FUNCTION_BLOCK FB_HE_SolidAttenuatorSlot EXTENDS FB_Fallible IMPLEMENTS I_HE_SolidAttenuatorSlot
VAR
    iFilter : I_HE_SolidAttenuatorFilter;
    eState : E_HE_SolidAttenuatorSlotState;
    bEnabled : BOOL;
END_VAR


METHOD FB_Init: BOOL
VAR_INPUT
    bInitRetains: BOOL; // TRUE: the retain variables are initialized (reset warm / reset cold)
    bInCopyCode: BOOL;  // TRUE: the instance will be copied to the copy code afterward (online change)

    Filter : I_HE_SolidAttenuatorFilter;
    State : E_HE_SolidAttenuatorSlotState;
    Enabled : BOOL;
END_VAR

iFilter := Filter;
eState := State;
bEnabled := Enabled;
END_METHOD


METHOD GetCenterPosition
VAR_INPUT
    CenterPosition : I_QuantityLREALPublic;
END_VAR

iFilter.GetCenterPosition(CenterPosition := CenterPosition);
END_METHOD


METHOD GetLength
VAR_INPUT
    Length : I_QuantityLREALPublic;
END_VAR

CASE eState OF
    E_HE_SolidAttenuatorSlotState.EMPTY:
        Length.Val := 0.0;
    E_HE_SolidAttenuatorSlotState.FULL:
        iFilter.GetLength(Length := Length);
END_CASE
END_METHOD


METHOD GetMaterial
VAR_IN_OUT
    Material : T_MaxString;
END_VAR

CASE eState OF
    E_HE_SolidAttenuatorSlotState.EMPTY:
        Material := '';
    E_HE_SolidAttenuatorSlotState.FULL:
        iFilter.GetMaterial(Material := Material);
END_CASE
END_METHOD


METHOD GetState : E_HE_SolidAttenuatorSlotState

GetState := eState;
END_METHOD


METHOD GetThicknessAt
VAR_INPUT
    QueryPointInAxisCoordinates : I_QuantityLREAL;
    Thickness : I_QuantityLREALPublic;
END_VAR

CASE eState OF
    E_HE_SolidAttenuatorSlotState.EMPTY:
        Thickness.Val := 0.0;
    E_HE_SolidAttenuatorSlotState.FULL:
        iFilter.GetThicknessAt(
            QueryPointInAxisCoordinates := QueryPointInAxisCoordinates,
            Thickness := Thickness
        );
END_CASE
END_METHOD


METHOD HasSpecifiedFilter : BOOL
VAR_INPUT
    Filter : I_HE_SolidAttenuatorFilter;
END_VAR

HasSpecifiedFilter := Filter = iFilter;
END_METHOD


METHOD IsEnabled : BOOL

IsEnabled := bEnabled;
END_METHOD

END_FUNCTION_BLOCK

(* stored: Version 1.1.0.1
   POU FB_HE_SolidAttenuatorSlot: Id {00460b56-1ea1-42cc-8f62-2eccd1d47e0f}, SpecialFunc None
   Method FB_Init: Id {58f02e95-764f-4ef9-819d-ad675cb7dc1c}
   Method GetCenterPosition: Id {6f9af3a0-1269-423f-a6cb-42e4f0745cf2}
   Method GetLength: Id {f422f0cc-ed5d-4a0b-834f-c85ec96acdff}
   Method GetMaterial: Id {c52d40a6-e5a0-408f-969b-1771f6a51579}
   Method GetState: Id {ec59714c-815d-4a33-9e3e-00e4b41216ef}
   Method GetThicknessAt: Id {735f6470-1a91-4cdc-9a90-02f3f22a622d}
   Method HasSpecifiedFilter: Id {d085ce8b-1fc7-41bf-ae9b-f79bec7fd4eb}
   Method IsEnabled: Id {06735b14-df5e-4a98-a89c-e5027127d234} *)
